PROGRAM POU
VAR
    bStart          : BOOL := TRUE;
    fbTimer         : TON;
    tTimerValue     : TIME := T#1S;
    fbTrigger       : R_TRIG;
    tTimeReturn1    : TIME;
    tTimeReturn2    : TIME;
    tDifference     : TIME;	
END_VAR

fbTimer(IN := bStart, PT := tTimerValue);
fbTrigger(CLK := fbTimer.IN);

IF fbTrigger.Q THEN
    tTimeReturn1  := TIME();
END_IF

IF fbTimer.Q THEN
    bStart        := FALSE;
    tTimeReturn2  := TIME();
    tDifference   := tTimeReturn2 - tTimeReturn1;    // The difference will be T#5s
END_IF

END_PROGRAM

(* stored: Version 1.1.0.1, ProductVersion 3.1.4024.9
   POU POU: Id {8accdd42-0350-4a26-b2f0-0849d5605925}, SpecialFunc None *)
